// TIA Portal V18 export
TYPE "PLCtoMES_AlarmExchange"
// stored: IsFailsafeCompliant false
   STRUCT
      "P-Alarm[X]" : Array[1..1024] of Bool;   // 设备报警映射区，PLC提供相应的报警说明表导入MES
      Reserve : Array[1..872] of Byte;   // 设备报警交互预留
   END_STRUCT;
END_TYPE
